{attribute 'GeneratedUsingTerminal: ELM9410-0000-0016'}
{attribute addProperty BoxType "ELM9410-0000-0016"}
{attribute addProperty Id "StatusAT %I*Status_F2CE6D917ValueAT %I*REAL4"}
{attribute addProperty CRC "1624595570"}
{attribute addProperty Size "11"}
TYPE MMS_Voltage_Us_In_Inputs_60D55C72 EXTENDS InputBase_8311D824 :
STRUCT
	{attribute addProperty Name "Status"}
	Status AT %I* : Status_F2CE6D91;
	{attribute addProperty Name "Value"}
	Value AT %I* : REAL;
END_STRUCT
END_TYPE

(* stored: Version 1.2.0.0, ProductVersion 3.1.4024.9
   DUT MMS_Voltage_Us_In_Inputs_60D55C72: Id {a5e8f3ee-c376-4c8e-b9d1-933dea7ee87d} *)
